// TIA Portal V19 export
DATA_BLOCK "PPrg_MAIN"   // DB98
{ DB_Accessible_From_OPC_UA := 'FALSE' }
// stored: DBAccessibleFromOPCUA false, MemoryReserve 100
   VAR
      PIVOT { ExternalAccessible := 'False'; ExternalVisible := 'False'; ExternalWritable := 'False'} : Array[1.."PPRG_TOTAL_ARCHIVE_ITEMS"] of "Prg_Pivot";
      GET_ITF { ExternalAccessible := 'False'; ExternalVisible := 'False'; ExternalWritable := 'False'} : "Prg_GetITF";
      RWD : Struct
         EMPTY { ExternalAccessible := 'False'; ExternalVisible := 'False'; ExternalWritable := 'False'} : "PPrg_Data";
         UPDATE { ExternalAccessible := 'False'; ExternalVisible := 'False'; ExternalWritable := 'False'} : "PPrg_Data";
         GET { ExternalAccessible := 'False'; ExternalVisible := 'False'; ExternalWritable := 'False'} : "PPrg_Data";
         HMI : "PPrg_Data";
         SCADA : "PPrg_Data";
      END_STRUCT;
      HMI : "Prg_HMI";
      SCADA : "Prg_SCADA";
   END_VAR
BEGIN
END_DATA_BLOCK
